{attribute 'qualified_only'}
{attribute 'strict'}
{attribute 'to_string'}
TYPE E_Motion :
(
	Sine,
	Ramp
);
END_TYPE

(* stored: Version 1.1.0.1, ProductVersion 3.1.4026.12
   DUT E_Motion: Id {650ba4e4-723b-42a7-941b-43686e73885b} *)
